PROGRAM pouS1Warnings
VAR
	
idbMsgWarn: FB_CheckMessageBounds;
END_VAR

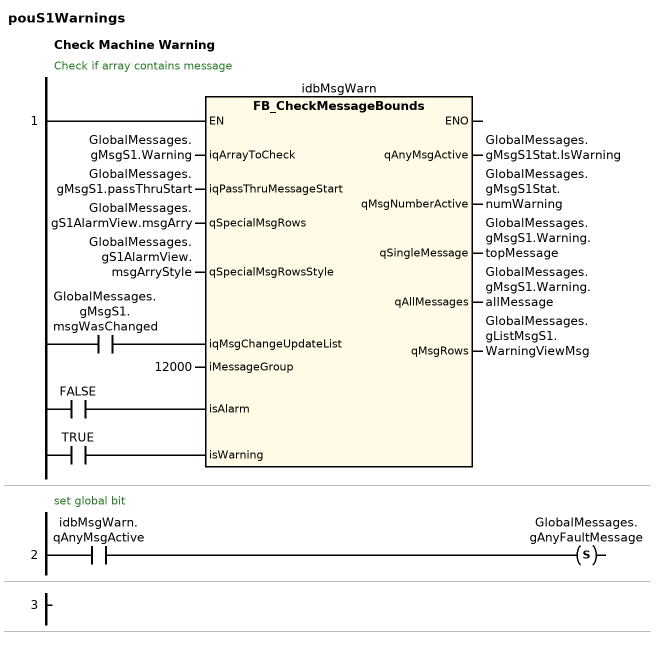
// NETWORK 1: Check Machine Warning
// Check if array contains message
idbMsgWarn(
    iqArrayToCheck := GlobalMessages.gMsgS1.Warning,
    iqPassThruMessageStart := GlobalMessages.gMsgS1.passThruStart,
    qSpecialMsgRows := GlobalMessages.gS1AlarmView.msgArry,
    qSpecialMsgRowsStyle := GlobalMessages.gS1AlarmView.msgArryStyle,
    iqMsgChangeUpdateList := GlobalMessages.gMsgS1.msgWasChanged,
    iMessageGroup := 12000,
    isAlarm := FALSE,
    isWarning := TRUE,
    qAnyMsgActive => GlobalMessages.gMsgS1Stat.IsWarning,
    qMsgNumberActive => GlobalMessages.gMsgS1Stat.numWarning,
    qSingleMessage => GlobalMessages.gMsgS1.Warning.topMessage,
    qAllMessages => GlobalMessages.gMsgS1.Warning.allMessage,
    qMsgRows => GlobalMessages.gListMsgS1.WarningViewMsg); // FB_CheckMessageBounds

// NETWORK 2
// set global bit
GlobalMessages.gAnyFaultMessage S= idbMsgWarn.qAnyMsgActive;

// NETWORK 3

END_PROGRAM

(* stored: Version 1.1.0.1, ProductVersion 3.1.4024.12
   POU pouS1Warnings: Id {65a0745a-e675-400f-ad40-91f4efb6ca28}, SpecialFunc None *)
